// Mitsubishi GX Works2 project: ZP_funtion_EX4   PLC: Q03UDV

PROGRAM MAIN
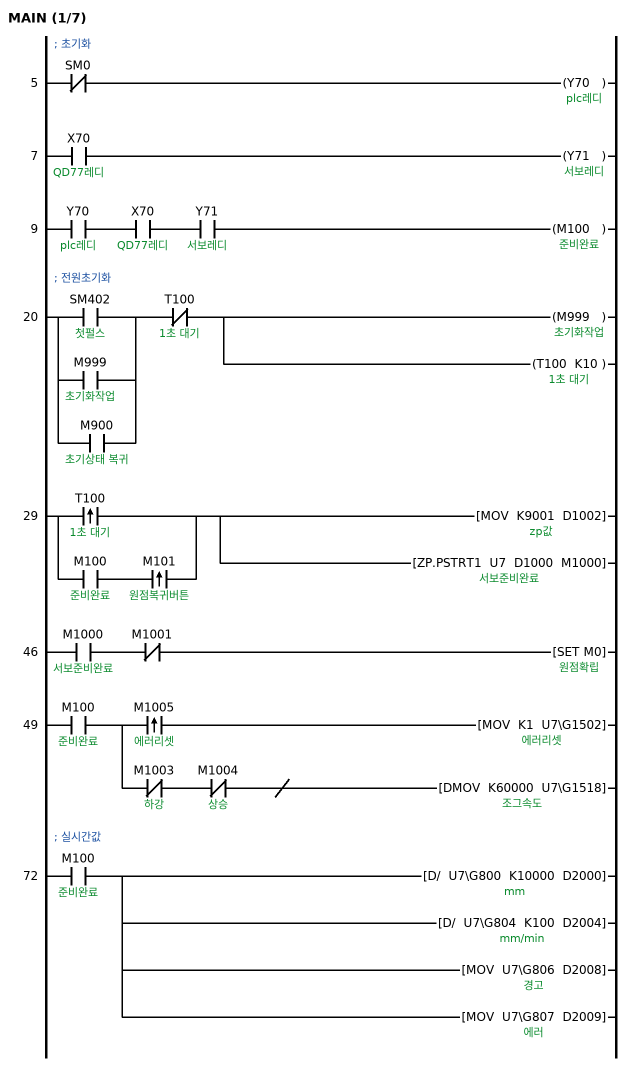
; 초기화
5     LDI     SM0
      OUT     Y70  ; plc레디
7     LD      X70  ; QD77레디
      OUT     Y71  ; 서보레디
9     LD      Y70  ; plc레디
      AND     X70  ; QD77레디
      AND     Y71  ; 서보레디
      OUT     M100  ; 준비완료
; 전원초기화
20    LD      SM402  ; 첫펄스
      OR      M999  ; 초기화작업
      OR      M900  ; 초기상태 복귀
      ANI     T100  ; 1초 대기
      OUT     M999  ; 초기화작업
      OUT     T100 K10  ; 1초 대기
29    LDP     T100  ; 1초 대기
      LD      M100  ; 준비완료
      ANDP    M101  ; 원점복귀버튼
      ORB
      MOV     K9001 D1002  ; zp값
      ZP.PSTRT1 U7 D1000 M1000  ; 서보준비완료
46    LD      M1000  ; 서보준비완료
      ANI     M1001
      SET     M0  ; 원점확립
49    LD      M100  ; 준비완료
      MPS
      ANDP    M1005  ; 에러리셋
      MOV     K1 U7\G1502  ; 에러리셋
      MPP
      ANI     M1003  ; 하강
      ANI     M1004  ; 상승
      INV
      DMOV    K60000 U7\G1518  ; 조그속도
; 실시간값
72    LD      M100  ; 준비완료
      D/      U7\G800 K10000 D2000  ; mm
      D/      U7\G804 K100 D2004  ; mm/min
      MOV     U7\G806 D2008  ; 경고
      MOV     U7\G807 D2009  ; 에러
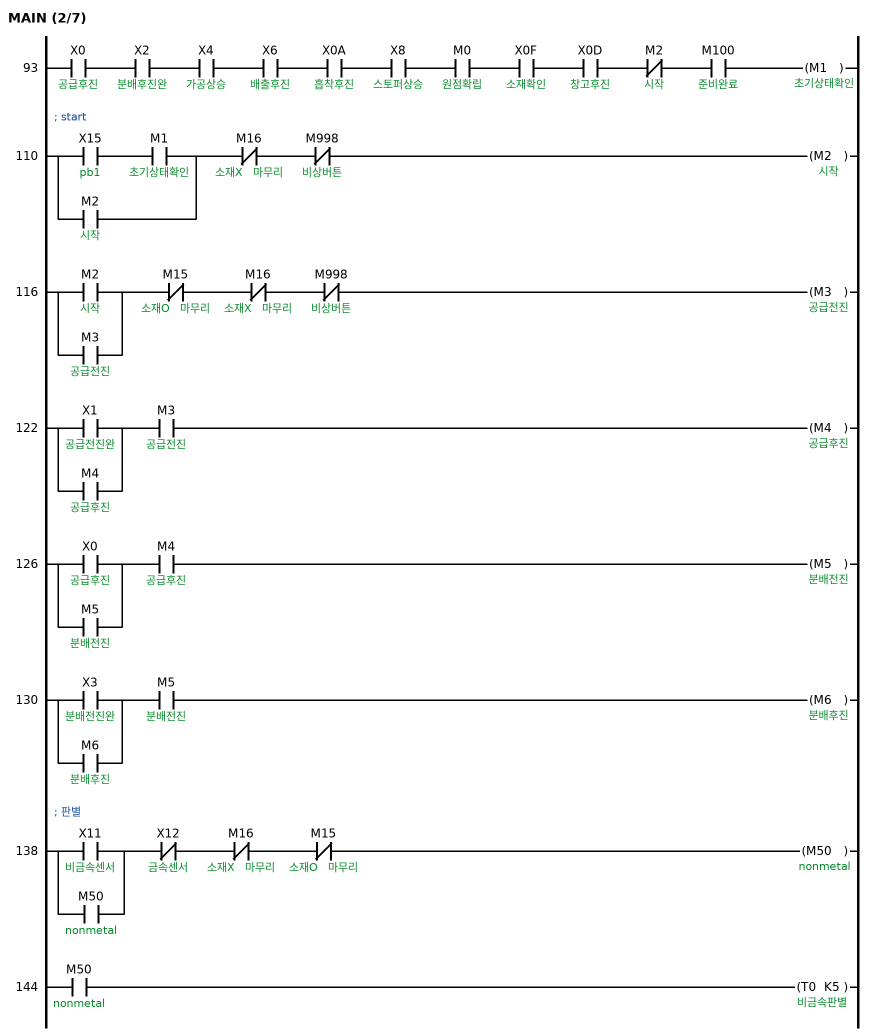
93    LD      X0  ; 공급후진
      AND     X2  ; 분배후진완
      AND     X4  ; 가공상승
      AND     X6  ; 배출후진
      AND     X0A  ; 흡착후진
      AND     X8  ; 스토퍼상승
      AND     M0  ; 원점확립
      AND     X0F  ; 소재확인
      AND     X0D  ; 창고후진
      ANI     M2  ; 시작
      AND     M100  ; 준비완료
      OUT     M1  ; 초기상태확인
; start
110   LD      X15  ; pb1
      AND     M1  ; 초기상태확인
      OR      M2  ; 시작
      ANI     M16  ; 소재X   마무리
      ANI     M998  ; 비상버튼
      OUT     M2  ; 시작
116   LD      M2  ; 시작
      OR      M3  ; 공급전진
      ANI     M15  ; 소재O   마무리
      ANI     M16  ; 소재X   마무리
      ANI     M998  ; 비상버튼
      OUT     M3  ; 공급전진
122   LD      X1  ; 공급전진완
      OR      M4  ; 공급후진
      AND     M3  ; 공급전진
      OUT     M4  ; 공급후진
126   LD      X0  ; 공급후진
      OR      M5  ; 분배전진
      AND     M4  ; 공급후진
      OUT     M5  ; 분배전진
130   LD      X3  ; 분배전진완
      OR      M6  ; 분배후진
      AND     M5  ; 분배전진
      OUT     M6  ; 분배후진
; 판별
138   LD      X11  ; 비금속센서
      OR      M50  ; nonmetal
      ANI     X12  ; 금속센서
      ANI     M16  ; 소재X   마무리
      ANI     M15  ; 소재O   마무리
      OUT     M50  ; nonmetal
144   LD      M50  ; nonmetal
      OUT     T0 K5  ; 비금속판별
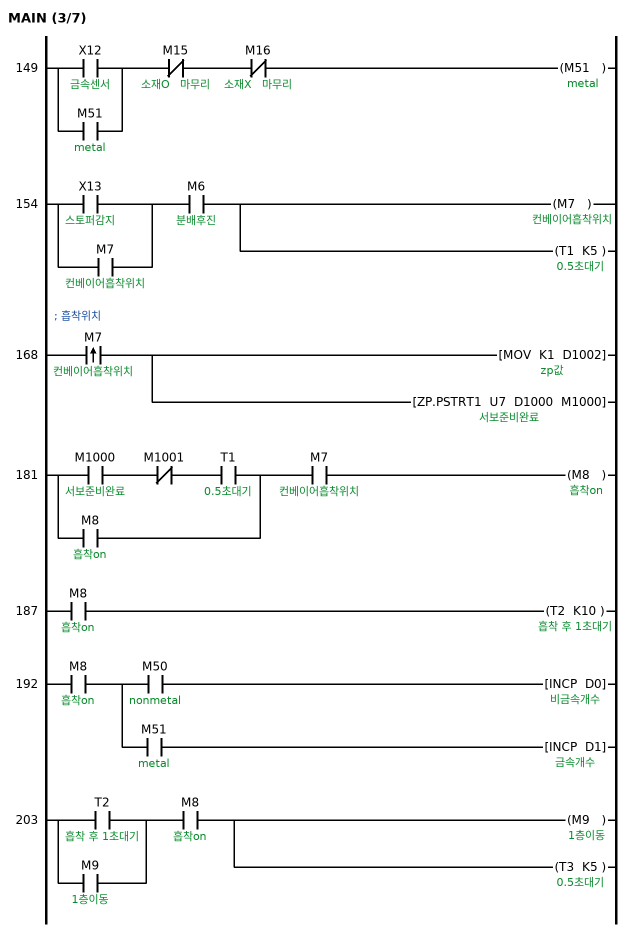
149   LD      X12  ; 금속센서
      OR      M51  ; metal
      ANI     M15  ; 소재O   마무리
      ANI     M16  ; 소재X   마무리
      OUT     M51  ; metal
154   LD      X13  ; 스토퍼감지
      OR      M7  ; 컨베이어흡착위치
      AND     M6  ; 분배후진
      OUT     M7  ; 컨베이어흡착위치
      OUT     T1 K5  ; 0.5초대기
; 흡착위치
168   LDP     M7  ; 컨베이어흡착위치
      MOV     K1 D1002
      ZP.PSTRT1 U7 D1000 M1000
181   LD      M1000  ; 서보준비완료
      ANI     M1001
      AND     T1  ; 0.5초대기
      OR      M8  ; 흡착on
      AND     M7  ; 컨베이어흡착위치
      OUT     M8  ; 흡착on
187   LD      M8  ; 흡착on
      OUT     T2 K10  ; 흡착 후 1초대기
192   LD      M8  ; 흡착on
      MPS
      AND     M50  ; nonmetal
      INCP    D0  ; 비금속개수
      MPP
      AND     M51  ; metal
      INCP    D1  ; 금속개수
203   LD      T2  ; 흡착 후 1초대기
      OR      M9  ; 1층이동
      AND     M8  ; 흡착on
      OUT     M9  ; 1층이동
      OUT     T3 K5  ; 0.5초대기
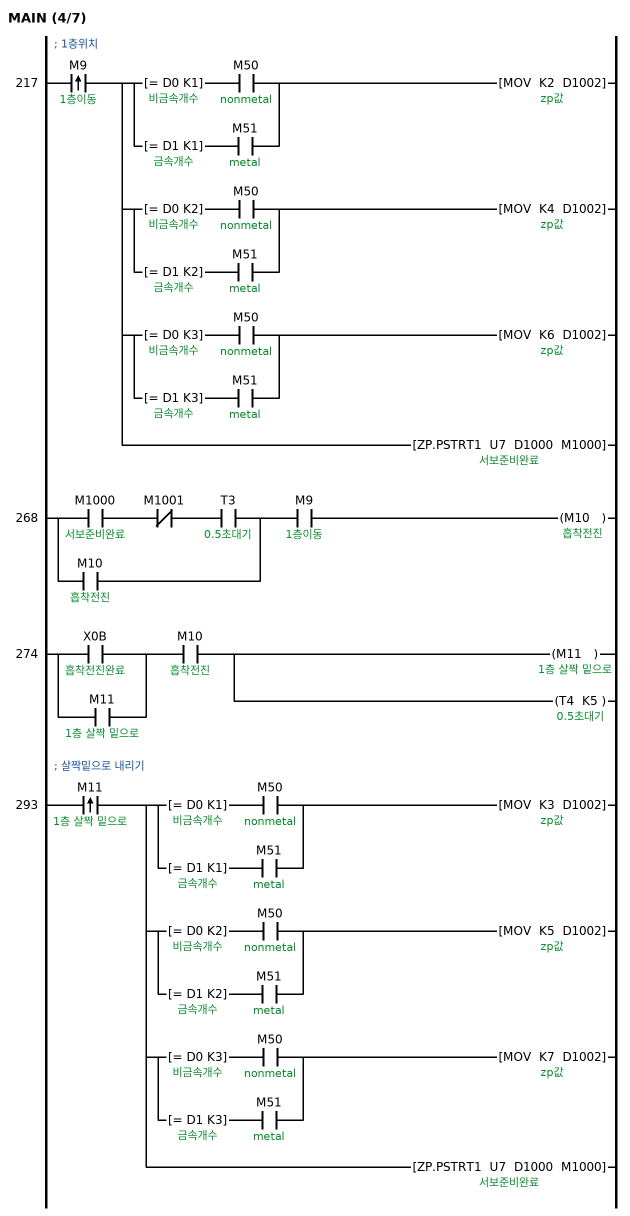
; 1층위치
217   LDP     M9  ; 1층이동
      MPS
      LD=     D0 K1  ; 비금속개수
      AND     M50  ; nonmetal
      LD=     D1 K1  ; 금속개수
      AND     M51  ; metal
      ORB
      ANB
      MOV     K2 D1002
      MRD
      LD=     D0 K2  ; 비금속개수
      AND     M50  ; nonmetal
      LD=     D1 K2  ; 금속개수
      AND     M51  ; metal
      ORB
      ANB
      MOV     K4 D1002
      MRD
      LD=     D0 K3  ; 비금속개수
      AND     M50  ; nonmetal
      LD=     D1 K3  ; 금속개수
      AND     M51  ; metal
      ORB
      ANB
      MOV     K6 D1002
      MPP
      ZP.PSTRT1 U7 D1000 M1000
268   LD      M1000  ; 서보준비완료
      ANI     M1001
      AND     T3  ; 0.5초대기
      OR      M10  ; 흡착전진
      AND     M9  ; 1층이동
      OUT     M10  ; 흡착전진
274   LD      X0B  ; 흡착전진완료
      OR      M11  ; 1층 살짝 밑으로
      AND     M10  ; 흡착전진
      OUT     M11  ; 1층 살짝 밑으로
      OUT     T4 K5  ; 0.5초대기
; 살짝밑으로 내리기
293   LDP     M11  ; 1층 살짝 밑으로
      MPS
      LD=     D0 K1  ; 비금속개수
      AND     M50  ; nonmetal
      LD=     D1 K1  ; 금속개수
      AND     M51  ; metal
      ORB
      ANB
      MOV     K3 D1002
      MRD
      LD=     D0 K2  ; 비금속개수
      AND     M50  ; nonmetal
      LD=     D1 K2  ; 금속개수
      AND     M51  ; metal
      ORB
      ANB
      MOV     K5 D1002
      MRD
      LD=     D0 K3  ; 비금속개수
      AND     M50  ; nonmetal
      LD=     D1 K3  ; 금속개수
      AND     M51  ; metal
      ORB
      ANB
      MOV     K7 D1002
      MPP
      ZP.PSTRT1 U7 D1000 M1000
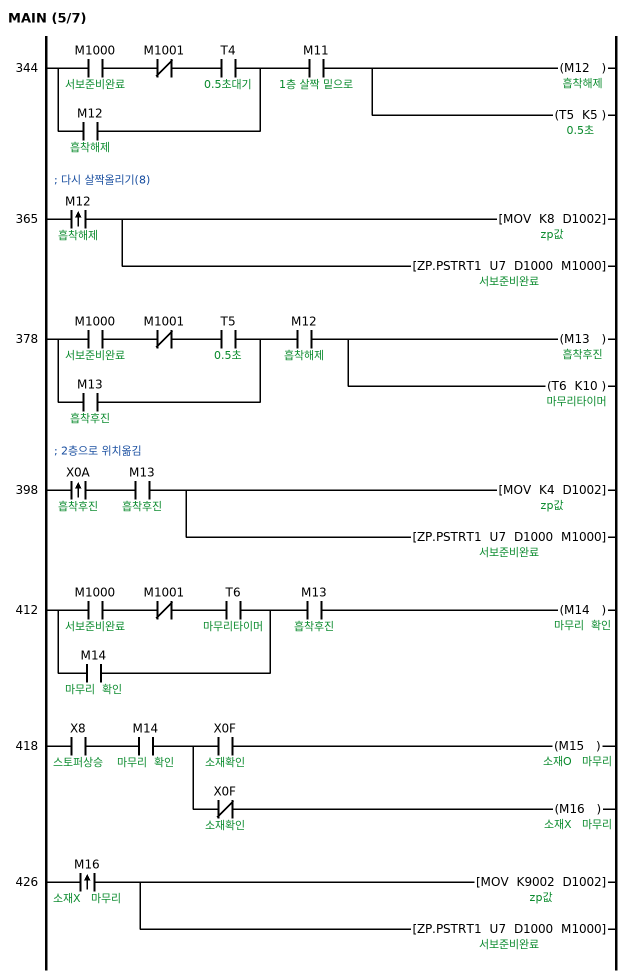
344   LD      M1000  ; 서보준비완료
      ANI     M1001
      AND     T4  ; 0.5초대기
      OR      M12  ; 흡착해제
      AND     M11  ; 1층 살짝 밑으로
      OUT     M12  ; 흡착해제
      OUT     T5 K5  ; 0.5초
; 다시 살짝올리기(8)
365   LDP     M12  ; 흡착해제
      MOV     K8 D1002
      ZP.PSTRT1 U7 D1000 M1000
378   LD      M1000  ; 서보준비완료
      ANI     M1001
      AND     T5  ; 0.5초
      OR      M13  ; 흡착후진
      AND     M12  ; 흡착해제
      OUT     M13  ; 흡착후진
      OUT     T6 K10  ; 마무리타이머
; 2층으로 위치옮김
398   LDP     X0A  ; 흡착후진
      AND     M13  ; 흡착후진
      MOV     K4 D1002
      ZP.PSTRT1 U7 D1000 M1000
412   LD      M1000  ; 서보준비완료
      ANI     M1001
      AND     T6  ; 마무리타이머
      OR      M14  ; 마무리  확인
      AND     M13  ; 흡착후진
      OUT     M14  ; 마무리  확인
418   LD      X8  ; 스토퍼상승
      AND     M14  ; 마무리  확인
      MPS
      AND     X0F  ; 소재확인
      OUT     M15  ; 소재O   마무리
      MPP
      ANI     X0F  ; 소재확인
      OUT     M16  ; 소재X   마무리
426   LDP     M16  ; 소재X   마무리
      MOV     K9002 D1002
      ZP.PSTRT1 U7 D1000 M1000
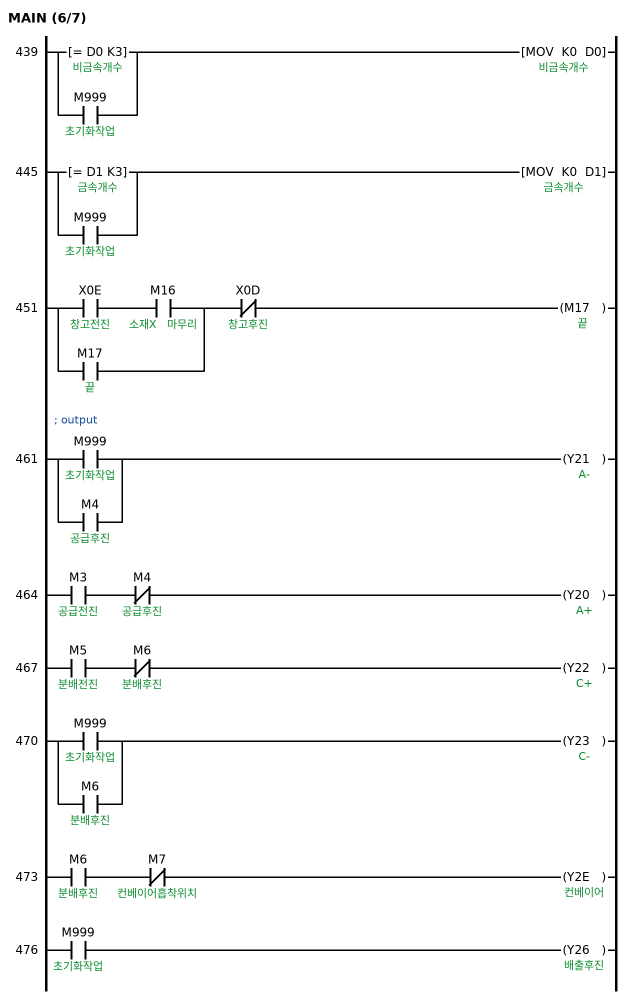
439   LD=     D0 K3  ; 비금속개수
      OR      M999  ; 초기화작업
      MOV     K0 D0
445   LD=     D1 K3  ; 금속개수
      OR      M999  ; 초기화작업
      MOV     K0 D1
451   LD      X0E  ; 창고전진
      AND     M16  ; 소재X   마무리
      OR      M17  ; 끝
      ANI     X0D  ; 창고후진
      OUT     M17  ; 끝
; output
461   LD      M999  ; 초기화작업
      OR      M4  ; 공급후진
      OUT     Y21  ; A-
464   LD      M3  ; 공급전진
      ANI     M4  ; 공급후진
      OUT     Y20  ; A+
467   LD      M5  ; 분배전진
      ANI     M6  ; 분배후진
      OUT     Y22  ; C+
470   LD      M999  ; 초기화작업
      OR      M6  ; 분배후진
      OUT     Y23  ; C-
473   LD      M6  ; 분배후진
      ANI     M7  ; 컨베이어흡착위치
      OUT     Y2E  ; 컨베이어
476   LD      M999  ; 초기화작업
      OUT     Y26  ; 배출후진
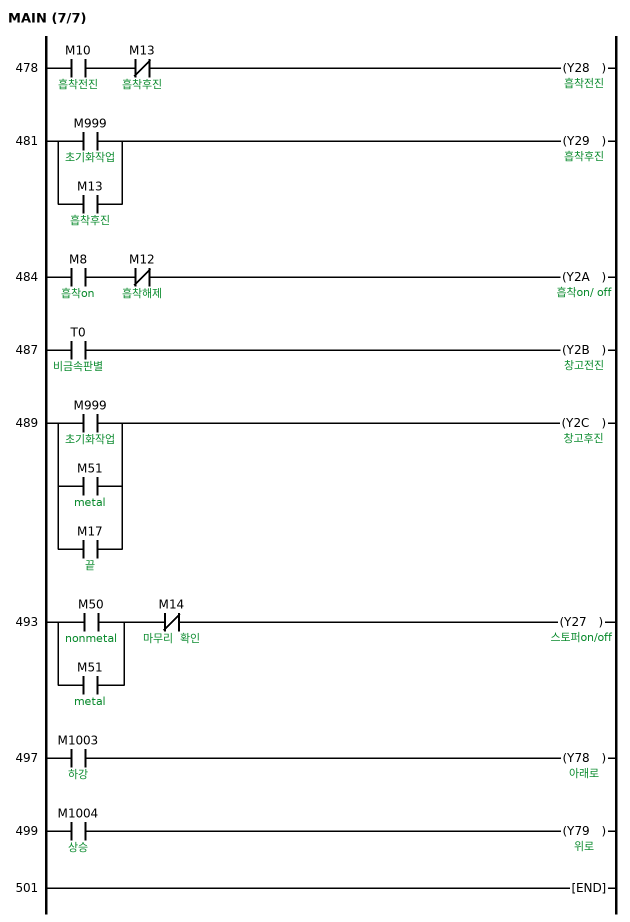
478   LD      M10  ; 흡착전진
      ANI     M13  ; 흡착후진
      OUT     Y28  ; 흡착전진
481   LD      M999  ; 초기화작업
      OR      M13  ; 흡착후진
      OUT     Y29  ; 흡착후진
484   LD      M8  ; 흡착on
      ANI     M12  ; 흡착해제
      OUT     Y2A  ; 흡착on/ off
487   LD      T0  ; 비금속판별
      OUT     Y2B  ; 창고전진
489   LD      M999  ; 초기화작업
      OR      M51  ; metal
      OR      M17  ; 끝
      OUT     Y2C  ; 창고후진
493   LD      M50  ; nonmetal
      OR      M51  ; metal
      ANI     M14  ; 마무리  확인
      OUT     Y27  ; 스토퍼on/off
497   LD      M1003  ; 하강
      OUT     Y78  ; 아래로
499   LD      M1004  ; 상승
      OUT     Y79  ; 위로
501   END
END_PROGRAM
